{attribute 'pack_mode' := '1'}  // needed for python pyads reading
TYPE ST_ProcessResult :
STRUCT
	
	Done:BOOL;
	OK:BOOL;
	Damage:BOOL;
	NOK:BOOL;
	NOK_Resaon: INT;
	
END_STRUCT
END_TYPE

(* stored: Version 1.1.0.1
   DUT ST_ProcessResult: Id {ec5c7ec2-883e-404f-a3f6-8d63ad30af4f} *)
